// TIA Portal project "FR" (V16)

(* hardware
DEVICE "S7-1200 station_1"  S7-1200 Station
   slot 0: "Rack_0"  S7-1200 Rack  Rack  V1.0
   slot 1: "PLC_1"  CPU 1212C AC/DC/Rly  6ES7 212-1BE40-0XB0  V4.4
*)

// ===== PLC "PLC_1"  CPU 1212C AC/DC/Rly =====

VAR_GLOBAL   // PLC tag table "Default tag table"
   "startf" AT %I0.0 : Bool;
   "stop" AT %I0.1 : Bool;
   "MOTOR1" AT %Q0.0 : Bool;
   "MOTOR2" AT %Q0.1 : Bool;
   "startb" AT %I0.2 : Bool;
   "Marker" AT %M0.0 : Bool;
   "TIMERON MARKER" AT %M0.1 : Bool;
   "TIMEROFF MARKER" AT %M0.2 : Bool;
   "COUNTER MARKER" AT %M0.3 : Bool;
   "MOTOR3" AT %M0.4 : Bool;
END_VAR

// folder: System blocks/Program resources

DATA_BLOCK "IEC_Timer_0_DB"   // DB1
{ S7_Optimized_Access := 'TRUE' }
AUTHOR : Simatic
FAMILY : IEC
NAME : IEC_TMR
VERSION : 1.0
// stored: InstanceOfName IEC_TIMER
"IEC_TIMER"
BEGIN
END_DATA_BLOCK

DATA_BLOCK "IEC_Counter_2_DB"   // DB2
{ S7_Optimized_Access := 'TRUE' }
AUTHOR : Simatic
FAMILY : IEC
NAME : CNTR
VERSION : 1.0
// stored: InstanceOfName IEC_COUNTER
"IEC_COUNTER"
BEGIN
END_DATA_BLOCK

DATA_BLOCK "IEC_Timer_1_DB_1"   // DB4
{ S7_Optimized_Access := 'TRUE' }
AUTHOR : Simatic
FAMILY : IEC
NAME : IEC_TMR
VERSION : 1.0
// stored: InstanceOfName IEC_TIMER
"IEC_TIMER"
BEGIN
END_DATA_BLOCK

// folder: (top level)

ORGANIZATION_BLOCK "Main"   // OB1, LAD, ProgramCycle
TITLE = "Main Program Sweep (Cycle)"
{ S7_Optimized_Access := 'TRUE' }
VERSION : 0.1
   VAR_INPUT
      Initial_Call : Bool;   // Initial call of this OB
      Remanence : Bool;   // =True, if remanent data are available
   END_VAR
BEGIN

REGION Network 1
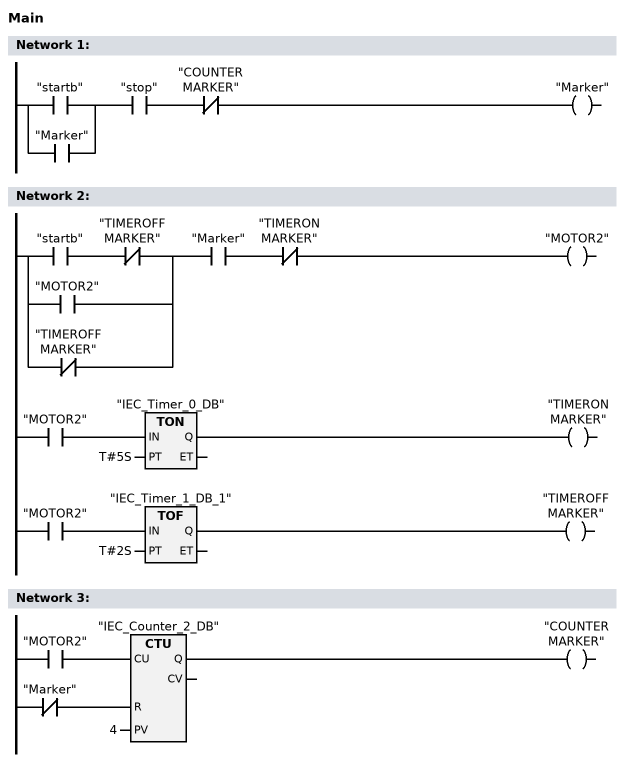
   RUNG wire#powerrail
      Contact( "startb" )
      wire#w1
      Contact( "stop" )
      I_Contact( "COUNTER MARKER" )
      Coil( "Marker" )
   END_RUNG
   RUNG wire#powerrail
      Contact( "Marker" )
   END_RUNG wire#w1
   // the same network as SCL:
   "Marker" := ("startb" OR "Marker") AND "stop" AND NOT "COUNTER MARKER";
END_REGION

REGION Network 2
   "MOTOR2" := (("startb" AND NOT "TIMEROFF MARKER") OR "MOTOR2" OR NOT "TIMEROFF MARKER") AND "Marker" AND NOT "TIMERON MARKER";
   "IEC_Timer_0_DB".TON(IN := "MOTOR2", PT := T#5S);
   "TIMERON MARKER" := "IEC_Timer_0_DB".Q;
   "IEC_Timer_1_DB_1".TOF(IN := "MOTOR2", PT := T#2S);
   "TIMEROFF MARKER" := "IEC_Timer_1_DB_1".Q;
END_REGION

REGION Network 3
   "IEC_Counter_2_DB".CTU(CU := "MOTOR2", R := NOT "Marker", PV := 4);
   "COUNTER MARKER" := "IEC_Counter_2_DB".Q;
END_REGION
END_ORGANIZATION_BLOCK